FUNCTION_BLOCK Step
VAR_INPUT
	iFaultCondition	: BOOL;
	iComplete		: BOOL;
	iRetry			: BOOL;
END_VAR

VAR_INPUT PERSISTENT
	cThisStep		: INT;
	cNextStep		: INT;
	cRecoveryStep	: INT;
	cTimeoutPreset	: TIME;
	cDescription	: STRING;
END_VAR

VAR_OUTPUT
	sActive			: BOOL;
	sFaulted		: BOOL;
	sTimedout		: BOOL;
	sComplete		: BOOL;
END_VAR

VAR_IN_OUT
	ioActiveStep	: INT;
END_VAR

VAR
	Status			: StatusStep;	
	ActiveTime		: TON;
END_VAR

ActiveTime.PT := cTimeoutPreset;

CASE Status OF
	StatusStep.Inactive:
							IF ioActiveStep = cThisStep THEN
								Status 			:= StatusStep.Active;
							END_IF
	StatusStep.Active:
							ActiveTime.IN 		:= TRUE;
							
							IF ActiveTime.Q THEN
								Status 			:= StatusStep.TimedOut;
								ActiveTime.IN 	:= FALSE;
							END_IF
							
							IF iFaultCondition THEN
								Status			:= StatusStep.Faulted;
							END_IF
							
							IF iComplete THEN
								Status			:= StatusStep.Complete;
							END_IF
	StatusStep.Faulted:
							IF iRetry THEN
								IF iFaultCondition = FALSE THEN
									Status			:= StatusStep.Active;
								ELSIF cRecoveryStep <> 0 THEN
									ioActiveStep := cRecoveryStep;
								END_IF
							END_IF
	StatusStep.TimedOut:
							IF iRetry THEN
								Status			:= StatusStep.Active;
							END_IF
	StatusStep.Complete:
							ioActiveStep := cNextStep;

END_CASE

END_FUNCTION_BLOCK

(* stored: Version 1.1.0.1, ProductVersion 3.1.4022.11
   POU Step: Id {efc0ed87-c022-492f-9b62-2f25b03d44fb}, SpecialFunc None *)
